Staubli VAL3: calcTool7En.pjx

--- calcTool7En.pjx ---
Parameters version=s7.3.1 stackSize=5000 millimeterUnit=true
Program file=example.pgx
Program file=language.pgx
Program file=mainCalcToolpp.pgx
Program file=readme.pgx
Program file=start.pgx
Program file=stop.pgx
Program file=usrButtonTxt.pgx
Data file=calcTool7En.dtx

--- calcTool7En.dtx ---
num nXPosButTxt[9]
  [2] = 5
  [3] = 10
  [4] = 15
  [5] = 20
  [6] = 25
  [7] = 30
  [8] = 35
num nYPosButTxt = 13
string sUsrMess[120]
  [0] = "Please select a language:"
  [1] = "Creation Tool complex"
  [2] = "This exercise requires:"
  [3] = "- A pointer attached"
  [4] = " to the robot's flange "
  [5] = "- A pointer placed as reference"
  [6] = " inside robot's working envelope "
  [7] = "- Your complex tool"
  [8] = "Press any key to continue..."
  [9] = "Creation of the reference tool"
  [10] = "Length of pointer (mm) :"
  [11] = "Mount the pointer on the robot's flange"
  [12] = "Go to the pointer placed as reference"
  [13] = "Press Enter"
  [14] = "when finish moving the robot"
  [15] = "Creation of your complex tool"
  [16] = "Mount your complex tool"
  [17] = "Go to the reference point "
  [18] = "Values of your tool :"
  [19] = "X :"
  [20] = "Y :"
  [21] = "Z :"
  [22] = "RX :"
  [23] = "RY :"
  [24] = "RZ :"
  [25] = "Verification of calculated TOOL"
  [26] = "Change to Tool mode"
  [27] = "  Select your tool "
  [28] = "Jog the robot in RX RY RZ"
  [29] = "in top of the reference pointer"
  [30] = "Press ESC if the result is not good"
  [31] = "Otherwise press ENTER"
  [32] = "Teaching finished !!!"
  [33] = "-END-"
  [41] = "Creation outil complexe"
  [42] = "Cette manipulation necessite :"
  [43] = "- Une pointe a fixer"
  [44] = " sur la bride du robot"
  [45] = "- Une contre-pointe a fixer"
  [46] = " dans l'enveloppe de travail du robot"
  [47] = "- Votre outil complexe"
  [48] = "Appui sur une touche pour continuer"
  [49] = "Creation de la pointe reference"
  [50] = "Longueur de la Pointe (mm) :"
  [51] = "Monter la pointe sur la bride du robot"
  [52] = "Allez sur la contre-pointe de reference"
  [53] = "Presser Enter"
  [54] = "quand la manipulation est terminee"
  [55] = "Creation de votre outil complexe"
  [56] = "Monter votre outil complexe"
  [57] = "Allez sur la pointe de reference"
  [58] = "Les cotes de votre outil :"
  [59] = "X : "
  [60] = "Y : "
  [61] = "Z : "
  [62] = "RX : "
  [63] = "RY : "
  [64] = "RZ : "
  [65] = "Verification du TOOL calcule"
  [66] = "Passer en mode TOOL"
  [67] = "Selectioner votre outil"
  [68] = "Faire des rotations RX RY RZ"
  [69] = "sur la contre-pointe"
  [70] = "Touche ESC si le resultat n'est pas bon"
  [71] = "Sinon touche ENTER"
  [72] = "L'apprentissage est terminΘ !!!"
  [73] = "-FIN-"
  [81] = "Calculo de herramienta compleja"
  [82] = "Este calculo requiere:"
  [83] = "- Una punta para fijar"
  [84] = "á en la brida del robot."
  [85] = "- Un contra-punta para fijar"
  [86] = "  sobre el area de trabajo del robot."
  [87] = "- La herramienta compleja."
  [88] = "Pulse cualquier tecla para continuar ..."
  [89] = "Creaci≤n herramienta de referencia"
  [90] = "Longitud de la punta (mm):"
  [91] = "Monte la punta en la brida del robot."
  [92] = "Ir a la contra-punta de referencia."
  [93] = "Pulse Intro"
  [94] = "  cuando la manipulaci≤n se acabe."
  [95] = "Creaci≤n de su herramienta compleja "
  [96] = "Ponga su herramienta compleja "
  [97] = "Ir hasta el punto de referencia."
  [98] = "Sφmbolos de la herramienta:"
  [99] = "X:"
  [100] = "Y:"
  [101] = "Z:"
  [102] = "RX:"
  [103] = "RY:"
  [104] = "RZ:"
  [105] = "Verificaci≤n Herramienta calculada"
  [106] = "Poner el robot en modo tool."
  [107] = "Seleccione su  herramienta."
  [108] = "Hacer rotaciones RX RY RZ"
  [109] = "  en la contra-punta"
  [110] = "ESC si el resultado no es correpto."
  [111] = "ENTER  si el resultado es correpto."
  [112] = "El calculo ha terminado!"
  [113] = "-FIN-"
tool tTool = {fatherId=flange[0], ioLink=valve1}

--- start.pgx ---
program start()
begin
  call example()
end

--- example.pgx ---
program example()
  local string l_sLanguage
begin
  //-----------------------------------------------------------------------
  //Header begin
  //Description of program
  //  This is an example of use of this library
  //  This program uses the following sub-programs :
  //  - language(): choose the language : "English", "French", "Spanish"
  //  - mainCalcToolpp(): calculates the tool transformation : a wizard will
  //  guide you thtough the steps.
  //History
  //  Creation : 08-04-08 - f.Rob
  //Header end
  //-----------------------------------------------------------------------

  //for choose the language
  call language(l_sLanguage)
  call mainCalcToolpp(l_sLanguage,tTool)
end

--- language.pgx ---
public program language(string& x_sLanguage[])
  local num l_nWhich
begin
  //-----------------------------------------------------------------------
  //Header begin
  //Description of program
  //  This program lets you choose the language : English, French or Spanish
  //
  //Input parameters
  //  string x_sLanguage :
  //    role : returns the language selected by the operator
  //    possible values : "English", "French" or "Spanish"
  //
  //History
  //  Creation : 08-04-08 - f.Rob
  //Header end
  //-----------------------------------------------------------------------

  userPage()
  cls()
  title("Language")
  gotoxy(7,10)
  put(sUsrMess[0])
  //Functions to display navigation keys (F1 through F8)
  //(here F2 "Engl", F4 "Fren" and F6 "Span")
  call usrButtonTxt(2,"Engl")
  call usrButtonTxt(4,"Fren")
  call usrButtonTxt(6,"Span")
  //
  //Waiting user choice 2 (F2) 4 (F4) or 6 (F6)
  do
    l_nWhich=(get()-270)
  until ((l_nWhich==2) or (l_nWhich==4) or (l_nWhich==6))
  //User choice : 2 (F2)=> English, 4 (F4)=> French, 6 (F6)=> Spanish
  switch l_nWhich
    case 2
      x_sLanguage="English"
    break
    case 4
      x_sLanguage="French"
    break
    case 6
      x_sLanguage="Spanish"
    break
  endSwitch
  cls()
end

--- mainCalcToolpp.pgx ---
public program mainCalcToolpp(string x_sLanguage, tool& x_tOutil[])
  local num l_nLongPointe
  local point l_pHere
  local point l_pRef
  local trsf l_trResultat
  local num l_nTouche
  local num l_nLanguage
  local tool l_tPointe
begin
  //-----------------------------------------------------------------------
  //Header begin
  //Description of program
  //  This program creates a tool using the pointer/counter pointer method
  //  A wizard will guide you through the steps
  //
  //Input parameters
  //  string x_sLanguage :
  //    role : defines the language GUI (Graphical User Interface) messages
  //
  //Output parameters
  //  tool& x_tOutil :
  //    role : calculated TCP (X, Y, Z, Rx, Ry, Rz)
  //
  //Example
  //  mainCalcToolpp(tPince,"French")
  //
  //History
  //  Creation : 08-04-08 - f.Rob
  //Header end
  //-----------------------------------------------------------------------

  //Initialization l_nTouche which allow to recovery keypresses
  l_nTouche=0
  userPage()
  //Test if there is no error in parameter language
  if (x_sLanguage=="English") or (x_sLanguage=="French") or (x_sLanguage=="Spanish")
    //Initialization l_nLanguage which allow to point in array  sUsrMess
    switch x_sLanguage
      case "English"
        l_nLanguage=0
      break
      case "French"
        l_nLanguage=40
      break
      case "Spanish"
        l_nLanguage=80
      break
    endSwitch
    //Displays instructions users (depend on the language)
    title(sUsrMess[1+l_nLanguage])
    cls()
    gotoxy(0,2)
    putln(sUsrMess[2+l_nLanguage])
    putln("")
    putln(sUsrMess[3+l_nLanguage])
    putln(sUsrMess[4+l_nLanguage])
    putln(sUsrMess[5+l_nLanguage])
    putln(sUsrMess[6+l_nLanguage])
    putln(sUsrMess[7+l_nLanguage])
    putln("")
    putln(sUsrMess[8+l_nLanguage])
    get()
    title(sUsrMess[9+l_nLanguage])
    l_tPointe=flange
    //For define length of the tool pointe (just axis z)
    do
      cls()
      l_nLongPointe=0
      gotoxy(0,3)
      put(sUsrMess[10+l_nLanguage])
      get(l_nLongPointe)
    until (l_nLongPointe>=0)
    l_tPointe.trsf={0,0,l_nLongPointe,0,0,0}
    //Displays instructions users (depend on the language)
    cls()
    gotoxy(0,3)
    putln(sUsrMess[11+l_nLanguage])
    putln(sUsrMess[12+l_nLanguage])
    putln("")
    putln(sUsrMess[13+l_nLanguage])
    putln(sUsrMess[14+l_nLanguage])
    //Waiting press enter to continue
    do
      l_nTouche=get()
    until (l_nTouche==270)
    //defines the reference point (on the counter-pointe)
    l_pRef=here(l_tPointe,world)
    cls()
    title(sUsrMess[15+l_nLanguage])
    gotoxy(0,3)
    putln(sUsrMess[16+l_nLanguage])
    putln(sUsrMess[4+l_nLanguage])
    do
      putln(sUsrMess[17+l_nLanguage])
      putln("")
      putln(sUsrMess[13+l_nLanguage])
      putln(sUsrMess[14+l_nLanguage])
      //Waiting press enter to continue
      do
        l_nTouche=get()
      until (l_nTouche==270)
      //Memorizing the reference point of your tool
      l_pHere=here(flange,world)
      //Creation of components of the tool
      x_tOutil.trsf=!l_pHere.trsf*(l_pRef.trsf)
      l_trResultat=x_tOutil.trsf
      //Displays components of the tool
      cls()
      title("")
      gotoxy(0,2)
      putln(sUsrMess[18+l_nLanguage])
      putln("")
      put(sUsrMess[19+l_nLanguage])
      putln(l_trResultat.x)
      put(sUsrMess[20+l_nLanguage])
      putln(l_trResultat.y)
      put(sUsrMess[21+l_nLanguage])
      putln(l_trResultat.z)
      put(sUsrMess[22+l_nLanguage])
      putln(l_trResultat.rx)
      put(sUsrMess[23+l_nLanguage])
      putln(l_trResultat.ry)
      put(sUsrMess[24+l_nLanguage])
      putln(l_trResultat.rz)
      putln("")
      putln(sUsrMess[13+l_nLanguage])
      //Waiting press enter to continue
      do
        l_nTouche=get()
      until (l_nTouche==270)
      //Explications for testing tool
      cls()
      title(sUsrMess[25+l_nLanguage])
      gotoxy(0,2)
      putln(sUsrMess[26+l_nLanguage])
      putln(sUsrMess[27+l_nLanguage])
      putln(sUsrMess[28+l_nLanguage])
      putln(sUsrMess[29+l_nLanguage])
      putln("")
      putln(sUsrMess[30+l_nLanguage])
      putln(sUsrMess[31+l_nLanguage])
      //If the user finds that the components are wrong
      //he press the ESC key (Back to learning reference point)
      l_nTouche=get()
      if !(l_nTouche==270)
        cls()
        gotoxy(0,3)
      endIf
    until (l_nTouche==270)
  else
    cls()
    title("Error")
    gotoxy(0,4)
    putln("Error language parameter !!!")
    putln("Press Enter to choose the language")
    //Waiting press enter to continue
    do
      l_nTouche=get()
    until (l_nTouche==270)
    call start()
  endIf
  cls()
  gotoxy(4,20)
  putln(sUsrMess[32+l_nLanguage])
  delay(2)
end

--- readme.pgx ---
program readme()
begin
  //Title: Calculates a tool transformation
  //
  //General description :
  //  This library calculates a tool transformation using the pointer/counter
  //  pointer method.
  //  1) Teach a reference point with an accurate tool. (calibrated pointer)
  //  2) Mount the tool and move the TCP (Tool center point) to the reference point
  //  The 6 components of the tool are calculated
  //
  //Hardware required :
  //  - Robot system    : any Staubli robot
  //  - Peripherals     : no peripherals required
  //
  //VAL3 options :
  //  - VAL3 version    : 7.3
  //  - VAL3 licenses   : no licenses required
  //  - VAL3 add-ons    : none
  //
  //Library version     : 7.3.1.0
  //
  //Public variables    : none
  //
  //Included libraries  : none
  //
  //Miscellaneous       : switched to version 7, IO library removed, no other modification - T.Caille 04/2012
  //
  //Keywords            : calculates, calcul, tool, outil, reference point, point de reference, components, composantes, pointer, pointe, counter pointer, contre pointe


end

--- stop.pgx ---
program stop()
begin
  waitEndMove()
  cls()
  title("")
  gotoxy(17,7)
  putln("-END-")
  resetMotion()
end

--- usrButtonTxt.pgx ---
program usrButtonTxt(num x_nWhichButton, string x_sButtonTxt)
begin
  //-----------------------------------------------------------------------
  //Header begin
  //Description of program
  //  This program lets you choose the key to display
  //
  //Input parameters
  //  num x_nWhichButton :
  //    role : choice of the navigation key
  //    possible values : 1 to 8 (F1 to F8)
  //
  //  string x_sButtonTxt :
  //    role : displays desired text
  //
  //History
  //  Creation : 08-04-08 - f.Rob
  //Header end
  //-----------------------------------------------------------------------

  //Position cursor X, Y
  gotoxy(nXPosButTxt[x_nWhichButton],nYPosButTxt)
  //Displays Text
  put(left(x_sButtonTxt,4))
  //Erases contents of text button parameters
  x_sButtonTxt=" "
end
